RoboDK station: Testing.rdk

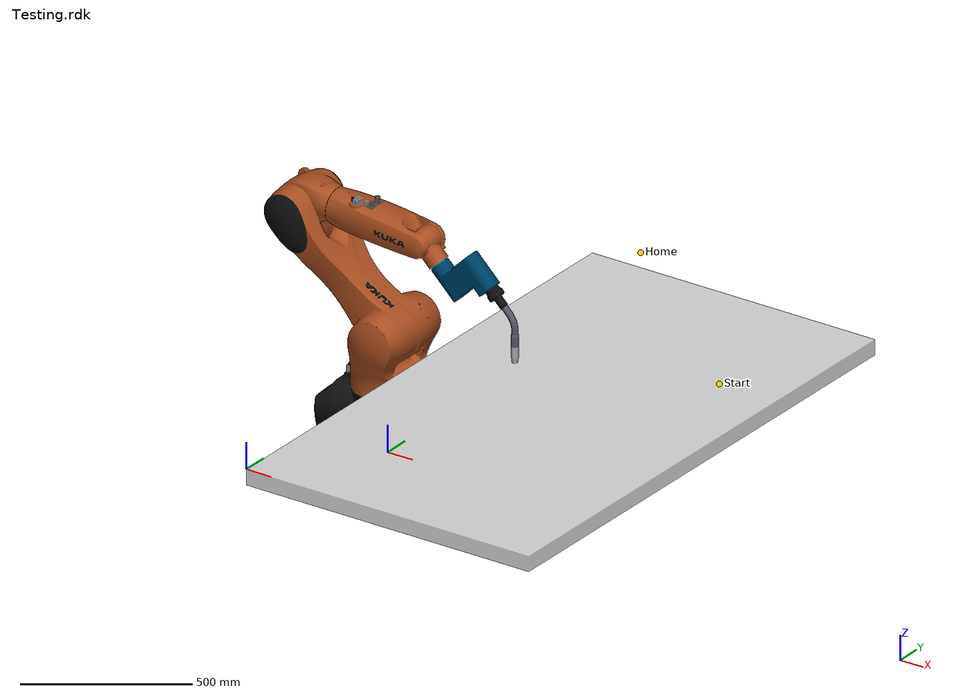
[picture v0: the station drawn from its stored meshes, robots at their saved joint values, targets as dots, program paths as lines]
Station Name (saved by RoboDK 5.2.1). Poses are relative to the parent item; angles as X-Y-Z fixed-axis rotations.
  - frame Frame object at (200, -1000, 400) mm
    - object Blackboard 250mm at (0, 0, 0) mm, size 250 x 250 x 50 mm
    - object Board at (0, 0, 0) mm, size 1000 x 1750 x 50 mm
  - frame KUKA KR 6 R900 sixx Base at (0, 0, 0) mm
    - robot KUKA KR 6 R900 sixx: 6 axes, payload 6 kg, reach 901 mm, repeatability 0.03 mm, weight 52 kg
        modified DH rows (alpha deg, a mm, theta deg, d mm): 0, 0, 0, 400; -90, 25, 0, 0; 0, 455, -90, 0; -90, 35, 0, 420; 90, 0, 0, 0; -90, 0, 180, 80
        joint limits [-170, -190, -120, -185, -120, -350] to [170, 45, 156, 185, 120, 350]; home [0, -90, 90, 0, 0, 0]; saved at [0, -134.393, 140.358, 0, 39.035, 0]
      - tool Weld gun, TCP at (-4, 0, 371.3) mm, rotated rx 0 ry 45 rz 0 deg, size 299.9 x 60 x 318.3 mm
    - target Home (Cartesian target) at (896.3, 0, 894) mm, rotated rx -180 ry 45 rz -180 deg; joints [0, -90, 90, 0, 0, 0] of KUKA KR 6 R900 sixx
    - target Start (Cartesian target) at (1000, 250, 400) mm, rotated rx 179.54 ry 0 rz 179.48 deg; joints [-20.268, -52.245, 62.928, 23.245, 38.494, -33.915] of KUKA KR 6 R900 sixx
  - Python program ListDrawing (listed below)

--- Python program ListDrawing ---
# Type help("robolink") or help("robodk") for more information
# Press F5 to run the script
# Documentation: https://robodk.com/doc/en/RoboDK-API.html
# Reference:     https://robodk.com/doc/en/PythonAPI/index.html
# Note: It is not required to keep a copy of this file, your python script is saved with the station
from robolink import *    # RoboDK API
from robodk import *      # Robot toolbox

# Notify user:
print('To edit this program:\nright click on the Python program, then, select "Edit Python script"')



list=[[900,250,400,-180,0,-180],
      [900,100,400,-180,0,-180],
      [1000,100,400,-180,0,-180],
      [1000,250,400,-180,0,-180],
      [850,250,600,-180,0,-180],
      [850,250,400,-180,0,-180],
      [550,250,400,-180,0,-180],
      [550,100,400,-180,0,-180],
      [850,100,400,-180,0,-180],
      [850,250,400,-180,0,-180],
      [750,250,400,-180,0,-180],
      [750,100,400,-180,0,-180],
      [650,100,400,-180,0,-180],
      [650,250,400,-180,0,-180],
      [550,250,400,-180,0,-180],

      [550,200,400,-180,0,-180],
      [450,250,400,-180,0,-180],
      [550,200,400,-180,0,-180],
      [550,150,400,-180,0,-180],
      [450,100,400,-180,0,-180],
      [450,100,600,-180,0,-180],
      [900,0,400,-180,0,-180],
      [900,-150,400,-180,0,-180],
      [450,-150,400,-180,0,-180],
      [500,-100,400,-180,0,-180],
      [450,-150,400,-180,0,-180],
      [900,-150,400,-180,0,-180],
      [900,-75,400,-180,0,-180],
      [1000,-90,400,-180,0,-180],
      [450,0,400,-180,0,-180]]


def drawing():

    for i in list:
     target=KUKA_2_Pose(i)
     print('target: '+str(i))
     robot.MoveL(target)





#---------------------------------------------------------------------------
# Program example:

#Program start
RDK = Robolink()

robot = RDK.Item('', ITEM_TYPE_ROBOT)
robot.setJoints([0,-90,90,0,0,0])        #set home position


# get the home target and the tool targets:
home = RDK.Item('Home')
Start = RDK.Item('Start')

# get the pose of the start (4x4 matrix representing position and orientation):
start_poseref = Start.Pose()

print(start_poseref)

#everytime restart from home and move to start point
framedraw=RDK.Item('Frame object')
robot.MoveJ(home)
robot.MoveJ(Start)
print('=====================================================================')

# delete previous image if any
image = RDK.Item('Board')
if image.Valid() and image.Type() == ITEM_TYPE_OBJECT: image.Delete()
#valid() check if the item is valid
#Type() return the type of item
#Delet() delet the item


# make a drawing board base on the object reference "Blackboard 250mm"
board_1m = RDK.Item('Blackboard 250mm')
board_1m.Copy()                    # Copy the item to the clipboard.
board_draw = framedraw.Paste()     # Paste the copied Item from the clipboard as a child of this item
board_draw.setVisible(True, False)
board_draw.setName('Board')
board_draw.Scale([4, 7, 1]) # adjust the board size to the image size (scale)

drawing()




raise Exception('Program not edited.')
